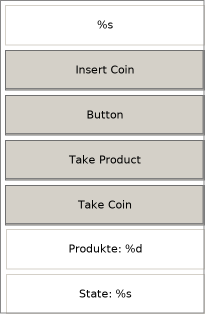
VISUALIZATION Panel  // 205x314
VAR_IN_OUT
	Panel		: POINTER TO ST_Panel;
END_VAR
    Button (5,50 200x40), "Insert Coin"
        tap Panel^.InsertCoin
    Textfield (5,5 200x40), "%s", text variable: Panel^.InstanzName
    Button (5,95 200x40), "Button"
        tap Panel^.Button
    Button (5,140 200x40), "Take Product"
        tap Panel^.TakeProduct
    Button (5,185 200x40), "Take Coin", text variable: Panel^.InstanzName
        tap Panel^.TakeCoin
    Textfield (6,229 199x40), "Produkte: %d", text variable: Panel^.NumberOfProducts
    Textfield (6,274 199x40), "State: %s", text variable: Panel^.State
END_VISUALIZATION

(* stored: Version 1.1.0.1, ProductVersion 3.1.4024.9
   Visu Panel: Id {ffbb87ac-5447-4e93-a8f1-5c683525b7ca} *)
